(* PLC project EFI, BrAutomation SafeDESIGNER  4.3.3.7 *)
(* stored: companyURL http://www.br-automation.com, creationDateTime Wed Mar 28 16:25:33 2018 *)

PROGRAM Main
  VAR  (* added by the conversion: wires and edge detectors of the diagram *)
    _AND_S747_OUT : ANY;
    _AND_S794_OUT : ANY;
    _SAFEBOOL_TO_BOOL796_OUT : BOOL;
    _AND_S673_OUT : ANY;
    _SAFEBOOL_TO_BOOL675_OUT : BOOL;
  END_VAR

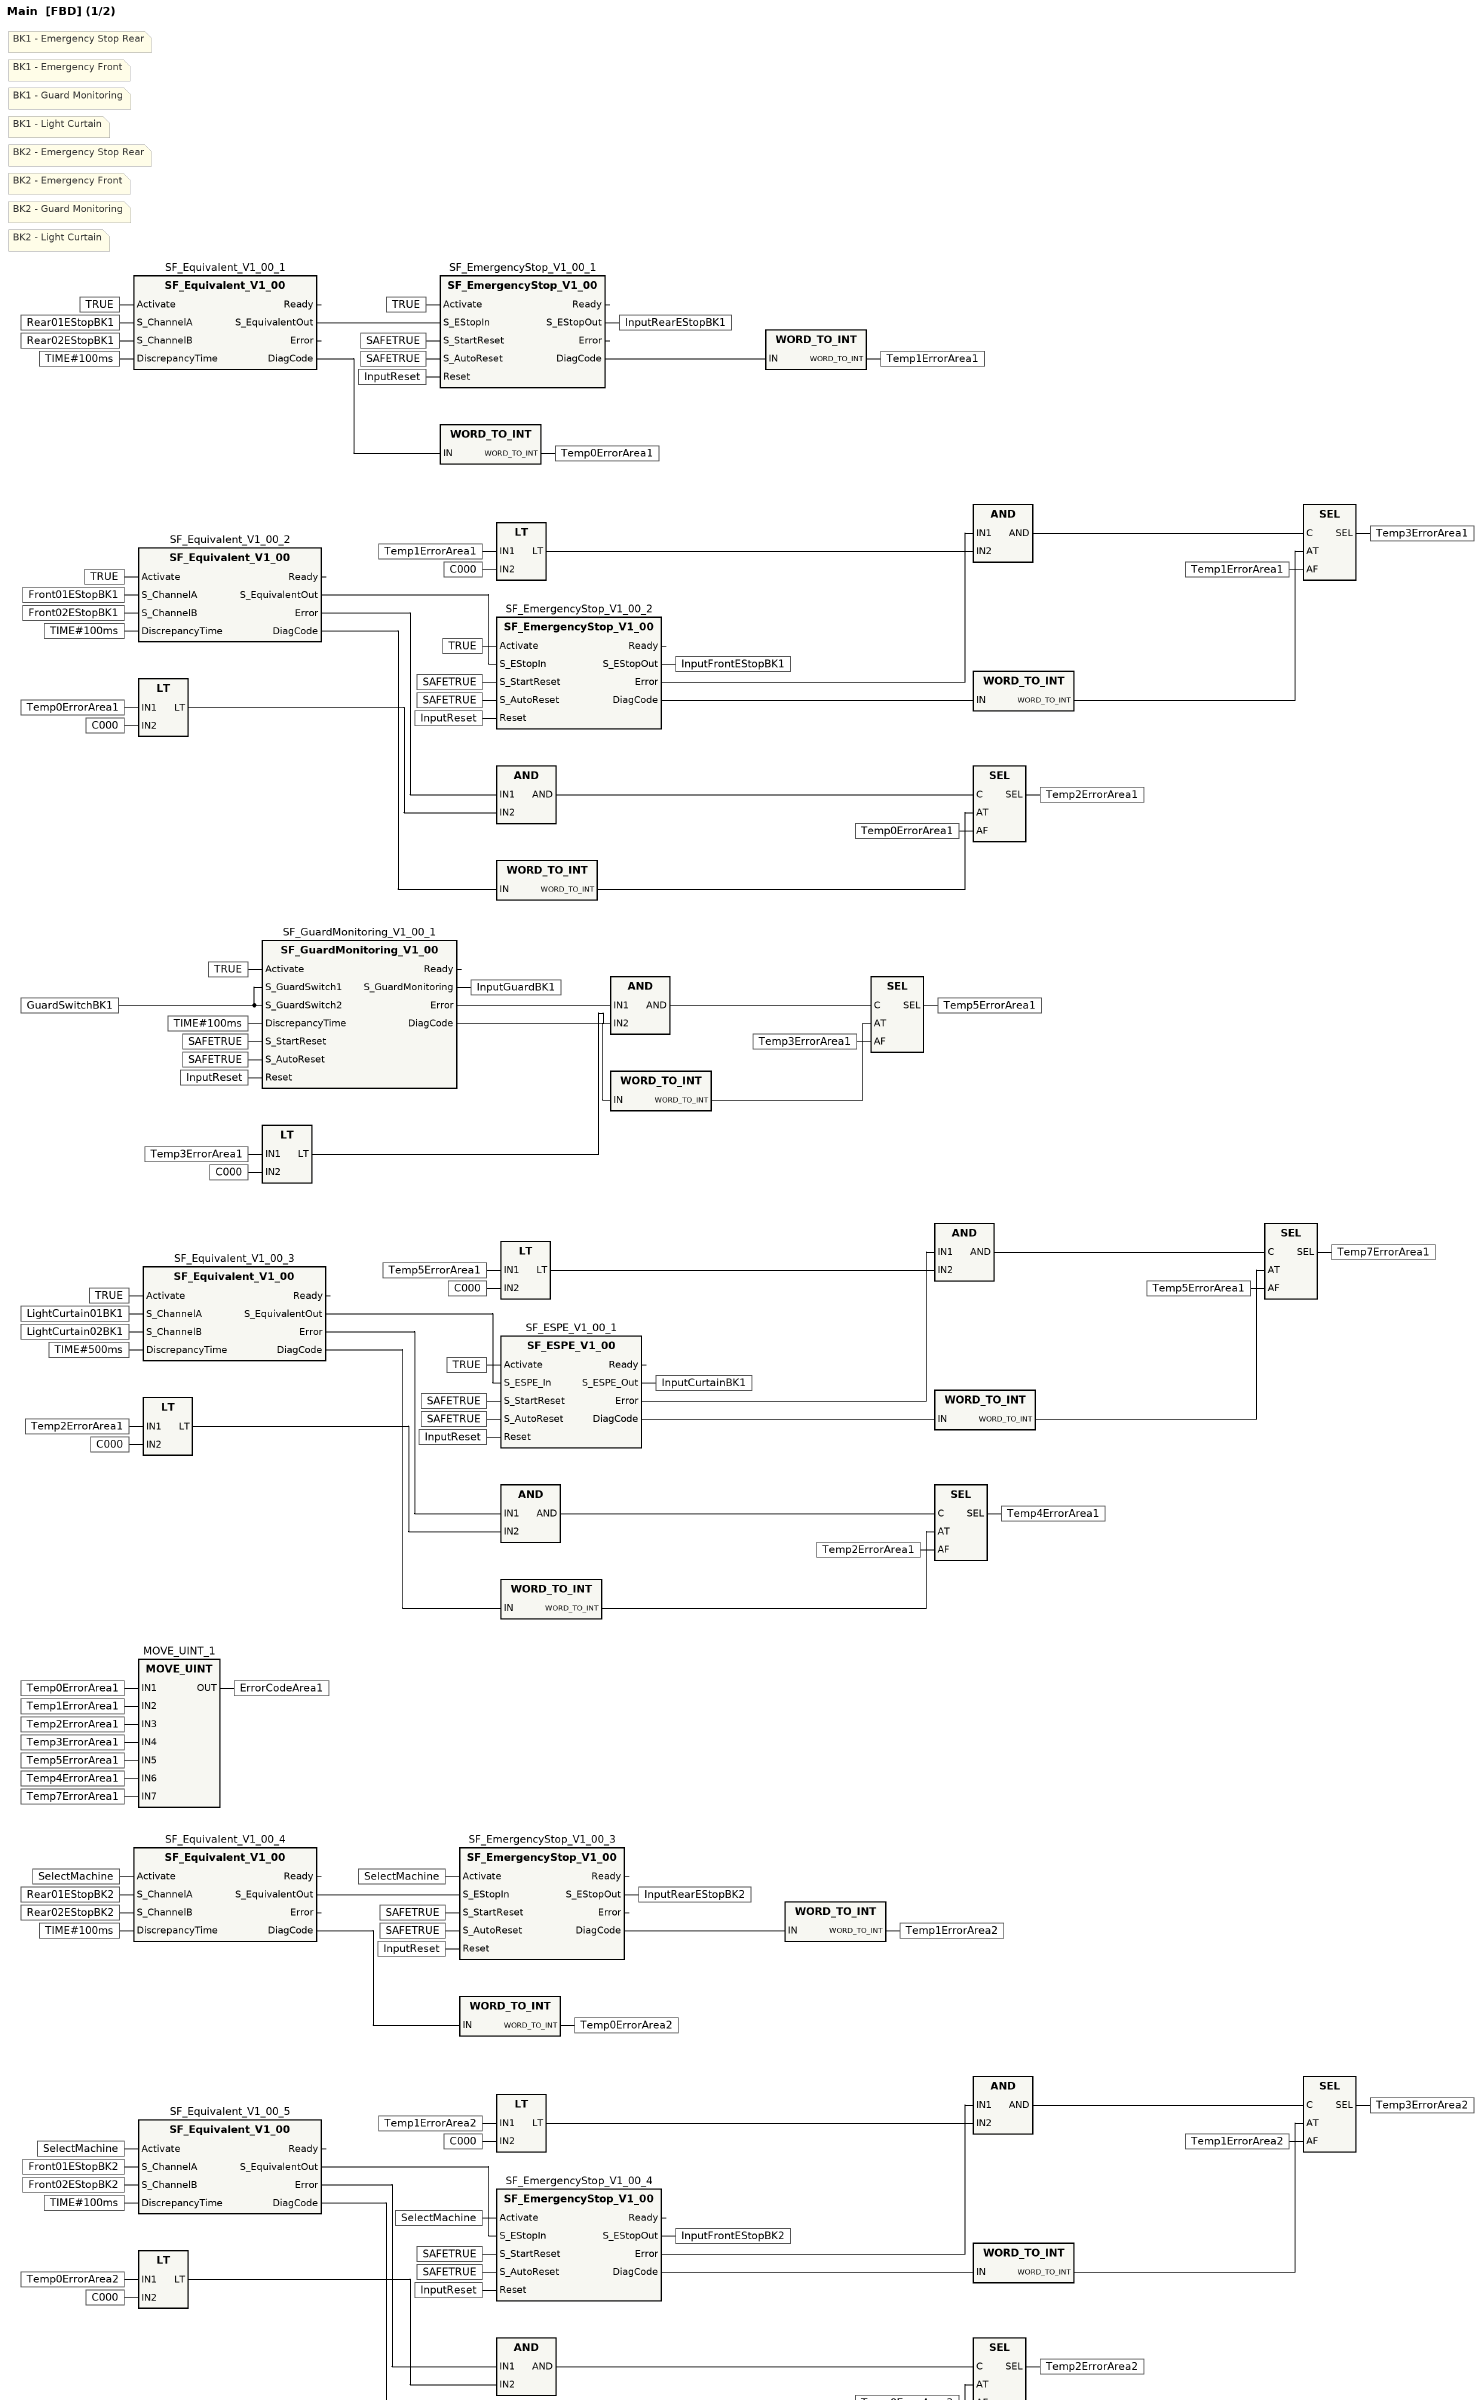
(* FBD diagram, written out as Structured Text *)
(* BK1 - Emergency Stop Rear *)
SF_Equivalent_V1_00_1(Activate := TRUE, S_ChannelA := Rear01EStopBK1, S_ChannelB := Rear02EStopBK1, DiscrepancyTime := TIME#100ms);
SF_EmergencyStop_V1_00_1(Activate := TRUE, S_EStopIn := SF_Equivalent_V1_00_1.S_EquivalentOut, S_StartReset := SAFETRUE, S_AutoReset := SAFETRUE, Reset := InputReset);
Temp1ErrorArea1 := WORD_TO_INT(SF_EmergencyStop_V1_00_1.DiagCode);
InputRearEStopBK1 := SF_EmergencyStop_V1_00_1.S_EStopOut;
Temp0ErrorArea1 := WORD_TO_INT(SF_Equivalent_V1_00_1.DiagCode);
(* BK1 - Emergency Front *)
SF_Equivalent_V1_00_2(Activate := TRUE, S_ChannelA := Front01EStopBK1, S_ChannelB := Front02EStopBK1, DiscrepancyTime := TIME#100ms);
SF_EmergencyStop_V1_00_2(Activate := TRUE, S_EStopIn := SF_Equivalent_V1_00_2.S_EquivalentOut, S_StartReset := SAFETRUE, S_AutoReset := SAFETRUE, Reset := InputReset);
InputFrontEStopBK1 := SF_EmergencyStop_V1_00_2.S_EStopOut;
Temp3ErrorArea1 := SEL(SF_EmergencyStop_V1_00_2.Error AND Temp1ErrorArea1 < C000, WORD_TO_INT(SF_EmergencyStop_V1_00_2.DiagCode), Temp1ErrorArea1);
Temp2ErrorArea1 := SEL(SF_Equivalent_V1_00_2.Error AND Temp0ErrorArea1 < C000, WORD_TO_INT(SF_Equivalent_V1_00_2.DiagCode), Temp0ErrorArea1);
(* BK1 - Guard Monitoring *)
SF_GuardMonitoring_V1_00_1(Activate := TRUE, S_GuardSwitch1 := GuardSwitchBK1, S_GuardSwitch2 := GuardSwitchBK1, DiscrepancyTime := TIME#100ms, S_StartReset := SAFETRUE, S_AutoReset := SAFETRUE, Reset := InputReset);
InputGuardBK1 := SF_GuardMonitoring_V1_00_1.S_GuardMonitoring;
Temp5ErrorArea1 := SEL(SF_GuardMonitoring_V1_00_1.Error AND Temp3ErrorArea1 < C000, WORD_TO_INT(SF_GuardMonitoring_V1_00_1.DiagCode), Temp3ErrorArea1);
(* BK1 - Light Curtain *)
SF_Equivalent_V1_00_3(Activate := TRUE, S_ChannelA := LightCurtain01BK1, S_ChannelB := LightCurtain02BK1, DiscrepancyTime := TIME#500ms);
SF_ESPE_V1_00_1(Activate := TRUE, S_ESPE_In := SF_Equivalent_V1_00_3.S_EquivalentOut, S_StartReset := SAFETRUE, S_AutoReset := SAFETRUE, Reset := InputReset);
InputCurtainBK1 := SF_ESPE_V1_00_1.S_ESPE_Out;
Temp7ErrorArea1 := SEL(SF_ESPE_V1_00_1.Error AND Temp5ErrorArea1 < C000, WORD_TO_INT(SF_ESPE_V1_00_1.DiagCode), Temp5ErrorArea1);
Temp4ErrorArea1 := SEL(SF_Equivalent_V1_00_3.Error AND Temp2ErrorArea1 < C000, WORD_TO_INT(SF_Equivalent_V1_00_3.DiagCode), Temp2ErrorArea1);
MOVE_UINT_1(IN1 := Temp0ErrorArea1, IN2 := Temp1ErrorArea1, IN3 := Temp2ErrorArea1, IN4 := Temp3ErrorArea1, IN5 := Temp5ErrorArea1, IN6 := Temp4ErrorArea1, IN7 := Temp7ErrorArea1);
ErrorCodeArea1 := MOVE_UINT_1.OUT;
(* BK2 - Emergency Stop Rear *)
SF_Equivalent_V1_00_4(Activate := SelectMachine, S_ChannelA := Rear01EStopBK2, S_ChannelB := Rear02EStopBK2, DiscrepancyTime := TIME#100ms);
SF_EmergencyStop_V1_00_3(Activate := SelectMachine, S_EStopIn := SF_Equivalent_V1_00_4.S_EquivalentOut, S_StartReset := SAFETRUE, S_AutoReset := SAFETRUE, Reset := InputReset);
InputRearEStopBK2 := SF_EmergencyStop_V1_00_3.S_EStopOut;
Temp0ErrorArea2 := WORD_TO_INT(SF_Equivalent_V1_00_4.DiagCode);
Temp1ErrorArea2 := WORD_TO_INT(SF_EmergencyStop_V1_00_3.DiagCode);
(* BK2 - Emergency Front *)
g_xInputSelectMachine := SelectMachine;
SF_Equivalent_V1_00_5(Activate := SelectMachine, S_ChannelA := Front01EStopBK2, S_ChannelB := Front02EStopBK2, DiscrepancyTime := TIME#100ms);
SF_EmergencyStop_V1_00_4(Activate := SelectMachine, S_EStopIn := SF_Equivalent_V1_00_5.S_EquivalentOut, S_StartReset := SAFETRUE, S_AutoReset := SAFETRUE, Reset := InputReset);
InputFrontEStopBK2 := SF_EmergencyStop_V1_00_4.S_EStopOut;
Temp3ErrorArea2 := SEL(SF_EmergencyStop_V1_00_4.Error AND Temp1ErrorArea2 < C000, WORD_TO_INT(SF_EmergencyStop_V1_00_4.DiagCode), Temp1ErrorArea2);
Temp2ErrorArea2 := SEL(SF_Equivalent_V1_00_5.Error AND Temp0ErrorArea2 < C000, WORD_TO_INT(SF_Equivalent_V1_00_5.DiagCode), Temp0ErrorArea2);
(* BK2 - Guard Monitoring *)
SF_GuardMonitoring_V1_00_2(Activate := SelectMachine, S_GuardSwitch1 := GuardSwitchBK2, S_GuardSwitch2 := GuardSwitchBK2, DiscrepancyTime := TIME#100ms, S_StartReset := SAFETRUE, S_AutoReset := SAFETRUE, Reset := InputReset);
InputGuardBK2 := SF_GuardMonitoring_V1_00_2.S_GuardMonitoring;
Temp5ErrorArea2 := SEL(SF_GuardMonitoring_V1_00_2.Error AND Temp3ErrorArea2 < C000, WORD_TO_INT(SF_GuardMonitoring_V1_00_2.DiagCode), Temp3ErrorArea2);
(* BK2 - Light Curtain *)
SF_Equivalent_V1_00_6(Activate := SelectMachine, S_ChannelA := LightCurtain01BK2, S_ChannelB := LightCurtain02BK2, DiscrepancyTime := TIME#500ms);
SF_ESPE_V1_00_2(Activate := SelectMachine, S_ESPE_In := SF_Equivalent_V1_00_6.S_EquivalentOut, S_StartReset := SAFETRUE, S_AutoReset := SAFETRUE, Reset := InputReset);
InputCurtainBK2 := SF_ESPE_V1_00_2.S_ESPE_Out;
Temp7ErrorArea2 := SEL(SF_ESPE_V1_00_2.Error AND Temp5ErrorArea2 < C000, WORD_TO_INT(SF_ESPE_V1_00_2.DiagCode), Temp5ErrorArea2);
Temp4ErrorArea2 := SEL(SF_Equivalent_V1_00_6.Error AND Temp2ErrorArea1 < C000, WORD_TO_INT(SF_Equivalent_V1_00_6.DiagCode), Temp2ErrorArea2);
MOVE_UINT_2(IN1 := Temp0ErrorArea2, IN2 := Temp1ErrorArea2, IN3 := Temp2ErrorArea2, IN4 := Temp3ErrorArea2, IN5 := Temp5ErrorArea2, IN6 := Temp4ErrorArea2, IN7 := Temp7ErrorArea2);
ErrorCodeArea2 := MOVE_UINT_2.OUT;
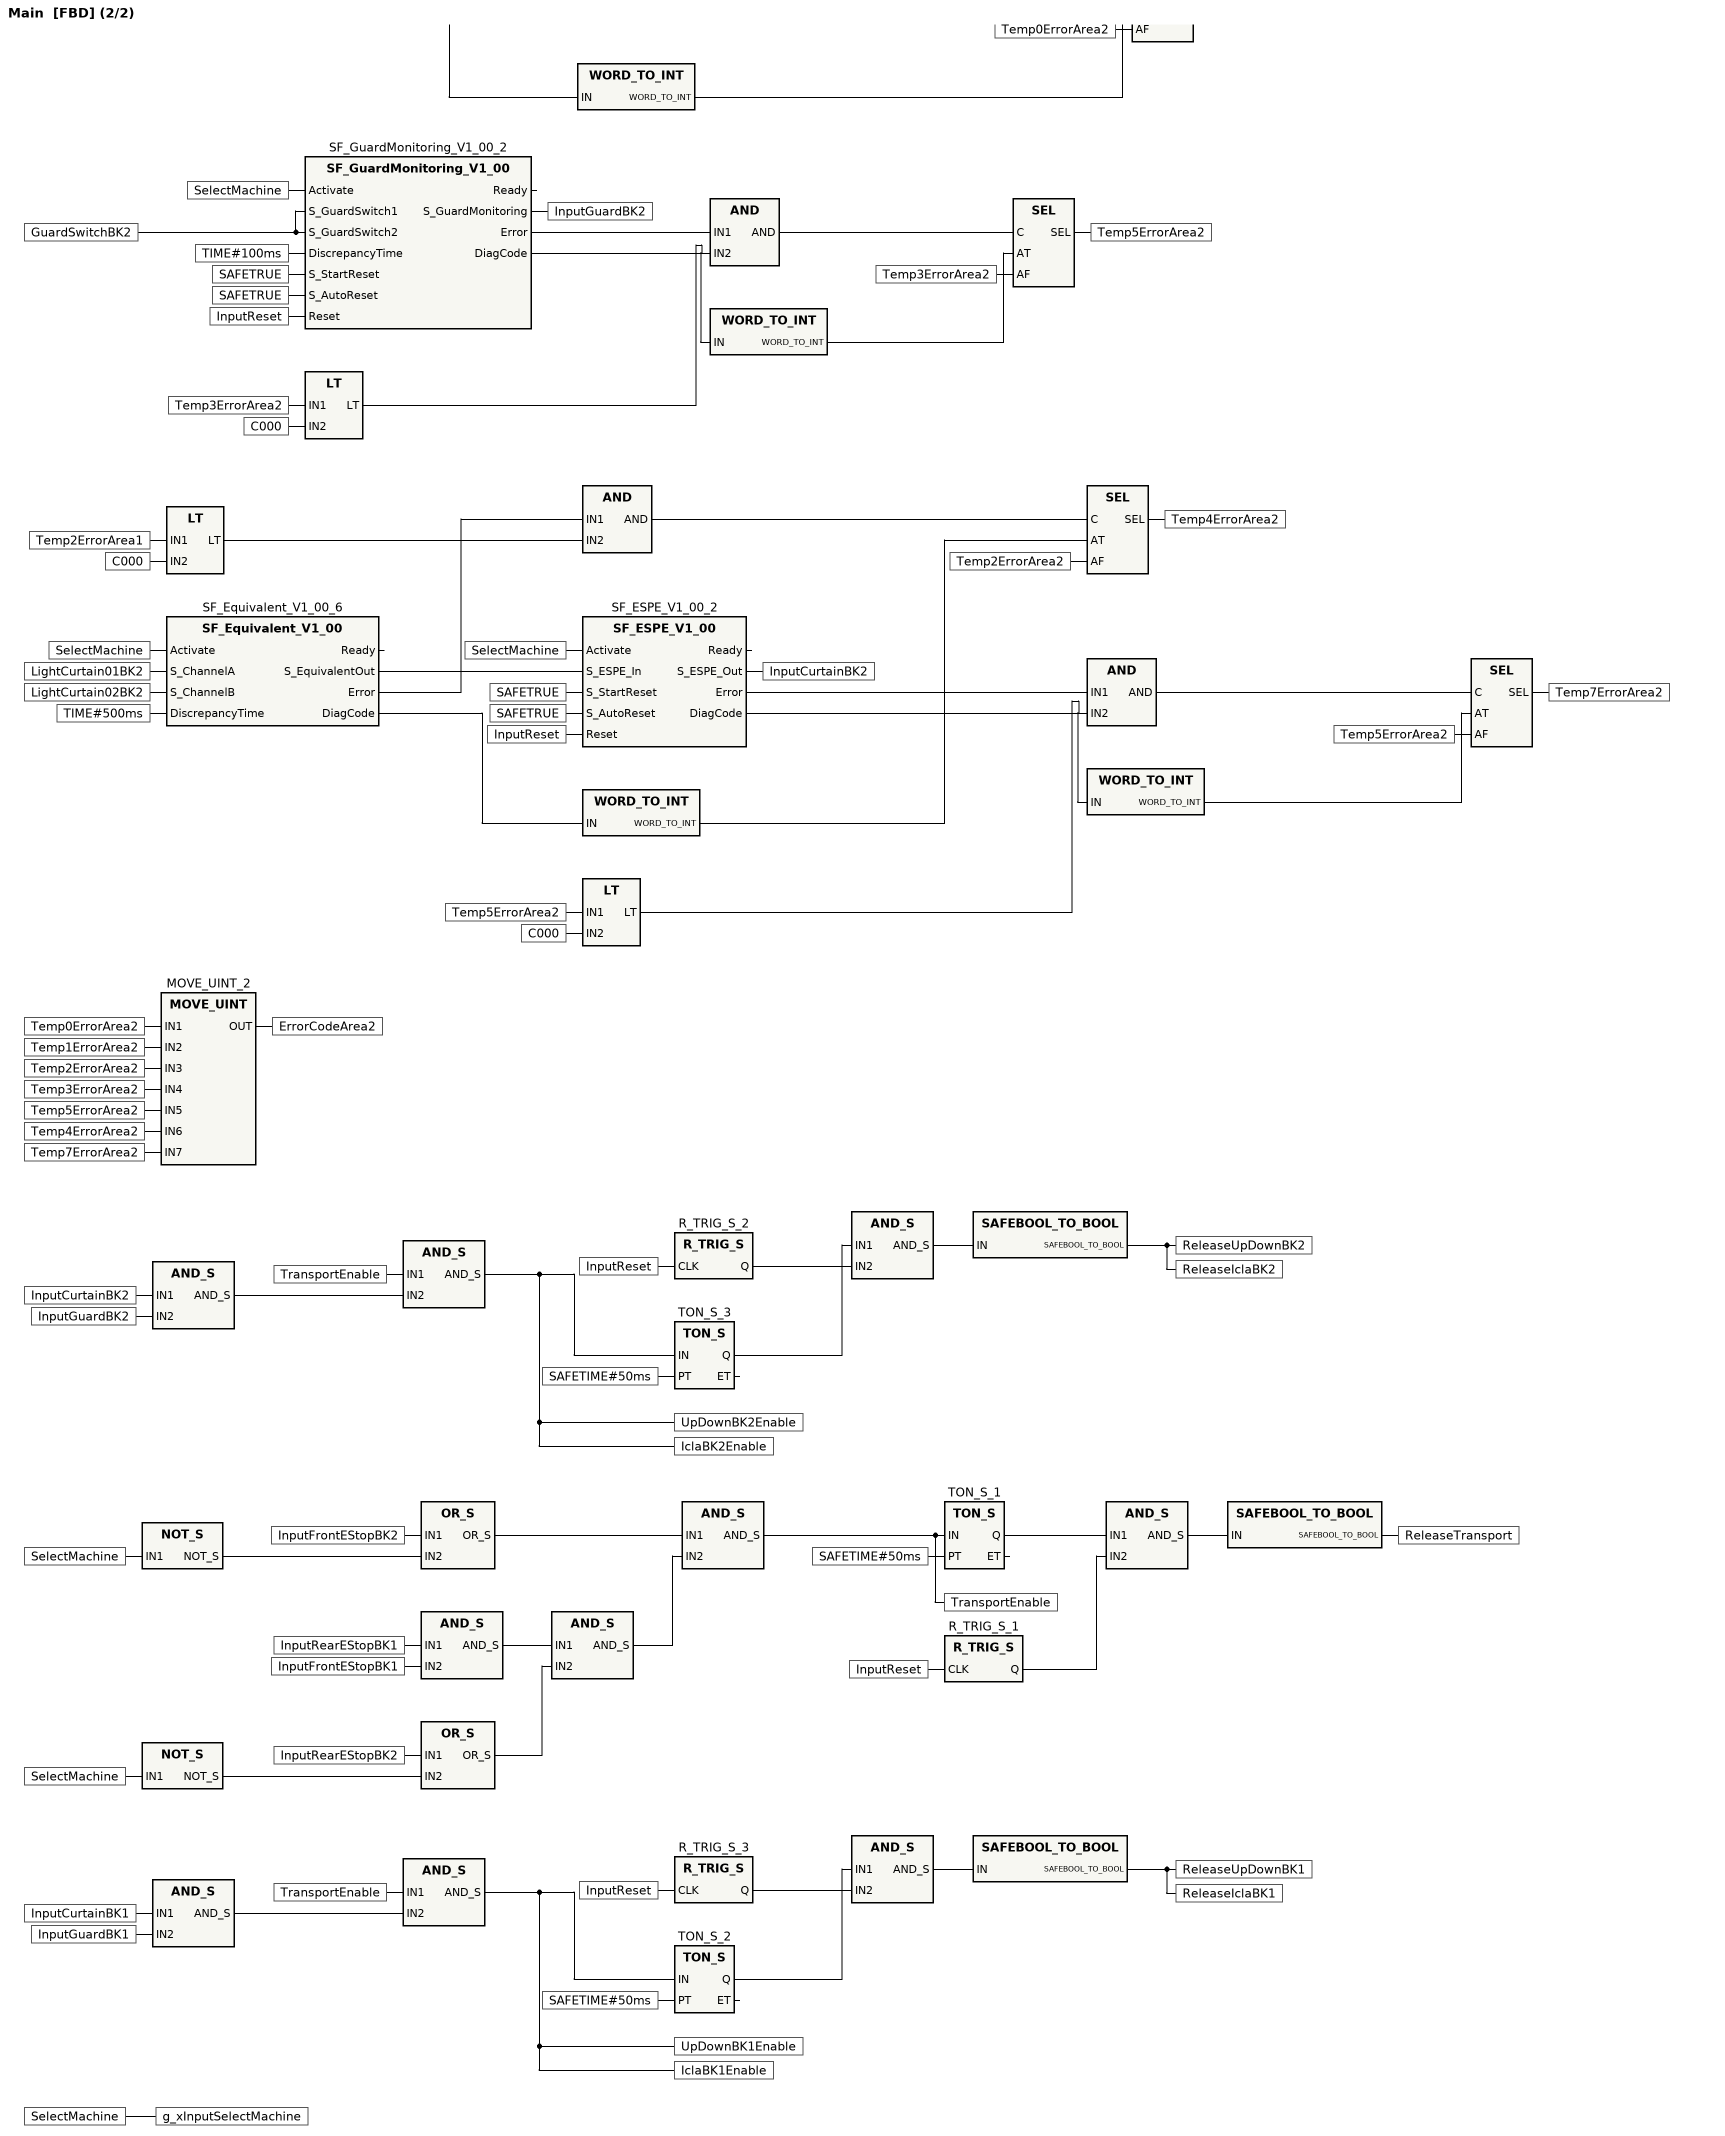
_AND_S747_OUT := AND_S(OR_S(InputFrontEStopBK2, NOT_S(SelectMachine)), AND_S(AND_S(InputRearEStopBK1, InputFrontEStopBK1), OR_S(InputRearEStopBK2, NOT_S(SelectMachine))));
TON_S_1(IN := _AND_S747_OUT, PT := SAFETIME#50ms);
R_TRIG_S_1(CLK := InputReset);
ReleaseTransport := SAFEBOOL_TO_BOOL(AND_S(TON_S_1.Q, R_TRIG_S_1.Q));
TransportEnable := _AND_S747_OUT;
_AND_S794_OUT := AND_S(TransportEnable, AND_S(InputCurtainBK1, InputGuardBK1));
UpDownBK1Enable := _AND_S794_OUT;
IclaBK1Enable := _AND_S794_OUT;
TON_S_2(IN := _AND_S794_OUT, PT := SAFETIME#50ms);
R_TRIG_S_3(CLK := InputReset);
_SAFEBOOL_TO_BOOL796_OUT := SAFEBOOL_TO_BOOL(AND_S(TON_S_2.Q, R_TRIG_S_3.Q));
ReleaseUpDownBK1 := _SAFEBOOL_TO_BOOL796_OUT;
ReleaseIclaBK1 := _SAFEBOOL_TO_BOOL796_OUT;
_AND_S673_OUT := AND_S(TransportEnable, AND_S(InputCurtainBK2, InputGuardBK2));
UpDownBK2Enable := _AND_S673_OUT;
IclaBK2Enable := _AND_S673_OUT;
TON_S_3(IN := _AND_S673_OUT, PT := SAFETIME#50ms);
R_TRIG_S_2(CLK := InputReset);
_SAFEBOOL_TO_BOOL675_OUT := SAFEBOOL_TO_BOOL(AND_S(TON_S_3.Q, R_TRIG_S_2.Q));
ReleaseUpDownBK2 := _SAFEBOOL_TO_BOOL675_OUT;
ReleaseIclaBK2 := _SAFEBOOL_TO_BOOL675_OUT;
END_PROGRAM
